// TIA Portal V16 export
// export: Created 2023-03-29T11:04:58.4849435Z, ExportSetting WithDefaults, DisplayName Totally Integrated Automation Portal, DisplayVersion V16 Update 6, DisplayName TIA Portal Version Control Interface, DisplayVersion V16 Update 2, DisplayName TIA Portal Openness, DisplayVersion V16 Update 6, DisplayName STEP 7 Professional, DisplayVersion V16 Update 6, DisplayName STEP 7 Safety, DisplayVersion V16, DisplayName WinCC Advanced, DisplayVersion V16 Update 6
DATA_BLOCK "dbControl press oxygen"   // DB64
AUTHOR : rtecmer
VERSION : 0.1
// stored: AutoNumber true, DBAccessibleFromOPCUA true, InstanceOfName Kontrola przekroczenia barMax, InstanceOfType FB
"Kontrola przekroczenia barMax"
   // VAR_INPUT
   //    dane_Pressure_bar : Real;
   //    Press_Max { ExternalAccessible := 'False'; ExternalVisible := 'False'; ExternalWritable := 'False'} : Real;
   // END_VAR
   // VAR_OUTPUT
   //    bar_max : Bool;
   // END_VAR
BEGIN
END_DATA_BLOCK
